// TIA Portal V20 export
// export: Created 2025-12-01T14:56:22.6342735Z, ExportSetting None, DisplayName Totally Integrated Automation Portal, DisplayVersion V20 Update 3, DisplayName TIA Portal Openness, DisplayVersion V20 Update 3, DisplayName TIA Portal Version Control Interface, DisplayVersion V20 Update 3, DisplayName STEP 7 Professional, DisplayVersion V20 Update 3, DisplayName STEP 7 Safety, DisplayVersion V20 Update 2, DisplayName WinCC Basic/Comfort/Advanced, DisplayVersion V20 Update 3, DisplayName WinCC Professional, DisplayVersion V20 Update 3, DisplayName WinCC Unified, DisplayVersion V20 Update 3
TYPE "EstadosMesa_Transporte_Paletizador_NDD"
   STRUCT
      Etapas_Reset : Bool;   // Etapa MESA en RESET
      Etapa_Vacia : Bool;   // Etapa MESA VACIA
      Etapa_Cargada : Bool;   // Etapa MESA CARGADA
      Etapas_Carga_E1 : Bool;   // Etapa CARGANDO MESA por E1
      Etapas_Descarga_S1 : Bool;   // Etapa DESCARGANDO MESA por S1
      Etapas_Carga_E2 : Bool;   // Etapa CARGANDO MESA por E2
      Etapas_Descarga_S2 : Bool;   // Etapa DESCARGANDO MESA por S2
      Etapas_Bloqueo : Bool;   // Etapa de BLOQUEO
      Descarga_Act : Bool;   // Memoria de DESCARGA ACTIVA
      Etapas_Carga_E0 : Bool;   // Etapa CARGANDO MESA por E0
      Etapas_Carga_E3 : Bool;   // Etapa CARGANDO MESA por E3
      Etapas_Descarga_S3 : Bool;   // Etapa DESCARGANDO MESA por S3
      Etapas_Carga_E4 : Bool;   // Etapa CARGANDO MESA por E4
      Etapas_Descarga_S4 : Bool;   // Etapa DESCARGANDO MESA por S4
      Etapas_Descarga_S0 : Bool;   // Etapa DESCARGANDO MESA por S0
      Manual : Bool;   // MESA EN MANUAL
      Err_Termico_E1_E3 : Bool;   // 01. TERMICO E1 E3
      Err_Termico_E2_E4 : Bool;   // 02. TERMICO E2 E4
      Err_Termico_Giro : Bool;   // 03. TERMICO GIRO
      Err_Mesa_Ocupada : Bool;   // 04. MESA OCUPADA
      Err_Perdida_PHs : Bool;   // 05. PERDIDA FOTOCELULA
      Err_TOut_Avance_E1_E3 : Bool;   // 06. TIMER TOUT Avance E1 E3
      Err_TOut_Retroceso_E1_E3 : Bool;   // 07. TIMER TOUT Retroceso E1 E3
      Err_TOut_Avance_E2_E4 : Bool;   // 08. TIMER TOUT Avance E2 E4
      Err_TOut_Retroceso_E2_E4 : Bool;   // 09. TIMER TOUT Retroceso E2 E4
      Err_TOut_Subir_TP_E1_E3 : Bool;   // 10. TIMER TOUT SUBIR TOPE E1 E3
      Err_TOut_Bajar_TP_E1_E3 : Bool;   // 11. TIMER TOUT BAJADA TOPE E1 E3
      Err_TOut_Subir_TP_E2_E4 : Bool;   // 12. TIMER TOUT SUBIDA TOPE E2 E4
      Err_TOut_Bajar_TP_E2_E4 : Bool;   // 13. TIMER TOUT BAJADA TOPE E2 E4
      Err_TOut_Bajada : Bool;   // 14. TIMER TOUT DE BAJADA DEL TRANSFER O MAQUETA
      Err_TOut_Subida : Bool;   // 15. TIMER TOUT DE SUBIDA DEL TRANSFER O MAQUETA
      Err_FTF_Sin_LibPHS_S1 : Bool;   // 16. FIN TRANSFER. SIN LIBERAR FOTOCELULA S1
      Err_FTF_Sin_LibPHS_S2 : Bool;   // 17. FIN TRANSFER. SIN LIBERAR FOTOCELULA S2
      Err_FTF_Sin_LibPHS_S3 : Bool;   // 18. FIN TRANSFER. SIN LIBERAR FOTOCELULA S3
      Err_FTF_Sin_LibPHS_S4 : Bool;   // 19. FIN TRANSFER. SIN LIBERAR FOTOCELULA S4
      Err_Salida_Lateral : Bool;   // 20. SALIDA LATERAL
      Err_Protusion : Bool;   // 21. PROTUSION
      Err_Interlock_Entrada : Bool;   // 22. INTERLOCK DE ENTRADA CON STV o VTD
      Err_Interlock_Salida : Bool;   // 23. INTERLOCK DE SALIDA CON STV o VTD
      Err_SegDescenso_EL : Bool;   // 24. DETECTOR DE DEGURIDAD EN DESCENSO DE LA MESA ELEVADORA
      Err_Tout_Giro : Bool;   // 25. TIMER TOUT DEL GIRO
      Err_Tout_Sacar : Bool;   // 26. TIMER TOUT DE SACRA LAS GARRAS
      Err_Tout_Recoger : Bool;   // 27. TIMER TOUT DE RECOGER LAS GARRAS
      Err_Tout_pos_0 : Bool;   // 28. TIMER TOUT DEL GIRO A 0º
      Err_Tout_pos_90 : Bool;   // 29. TIMER TOUT DEL GIRO A 90º
      Err_pHs_Galibo : Bool;   // 30. ERROR DE FOCELULAS DE GALIBO
      Err_DetectorTRANSFER : Bool;   // 31. ERROR DE DETECCION DEL TRANSFER ELECTRICO
      Err_Termico_elevacion : Bool;   // 32. ERROR TERMICO EN EL TRANSFER ELECTRICO
      Err_Nodo_SSCC : Bool;   // 33. ERROR PERDIDA NODO DEL SCANNER
      Err_SSCC_LectPorcentaje : Bool;   // 34. ERROR PORCENTAJE DE LECTURAS DE ESCANNER
      Err_SSCC_LectConsecutiva : Bool;   // 35. ERROR LECTURAS DE ESCANER CONSECUTICAS
      Err_MaquinaAsociada : Bool;   // 36. ERROR MAQUINA ASOCIADA A LA MESA
      Err_Extradimensiones : Bool;   // 37. ERROR PALETA FLEJADA
      Err_EnviadoPorJDT : Bool;   // 38. ERROR ENVIADO POR EL JDT
      Err_DatosPLC : Bool;   // 39. ERROR DE DATOS DEL PLC
      Error_Mx : Bool;   // Marca General Error
      En_Termico1 : Bool;   // Entrada de TERMICO 1
      En_Termico2 : Bool;   // Entrada de TERMICO 2
      En_PHS_1 : Bool;   // Entrada de FOTOCELULA 1
      En_PHS_2 : Bool;   // Entrada de FOTOCELULA 2
      En_Transfer_UP : Bool;   // Entrada TRANSFER/MAQUETA/MESA ELEVADORA ARRIBA
      En_Transfer_DOWN : Bool;   // Entrada TRANSFER/MAQUETA/MESA ELEVADORA ABAJO
      En_Tope1_UP : Bool;   // Entrada TOPE 1 ARRIBA
      En_Tope1_DOWN : Bool;   // Entrada TOPE 1 ABAJO
      En_Tope2_UP : Bool;   // Entrada TOPE 2 ARRIBA
      En_Tope2_DOWN : Bool;   // Entrada TOPE 2 ABAJO
      En_PHS_3 : Bool;   // Entrada de FOTOCELULA 3
      En_PHS_4 : Bool;   // Entrada de FOTOCELULA 4
      En_PHS_5 : Bool;   // Entrada de FOTOCELULA 5
      En_Giro_270 : Bool;   // …
      En_pHs_Prot1 : Bool;   // Entrada PROTUSION 1
      En_Detector_carretilla : Bool;   // Entrada detector de carretilla
      En_Giro_0 : Bool;   // Entrada Giro pos 0
      En_Giro_90 : Bool;   // Entrada Giro pos 90
      En_Giro_180 : Bool;   // Entrada Giro pos 180
      En_pHs_Prot2 : Bool;   // Entrada PROTUSION 2
      En_pHs_Prot3 : Bool;   // Entrada PROTUSION 3
      En_pHs_Prot4 : Bool;   // Entrada PROTUSION 4
      En_Empuj_Extendido : Bool;   // Entrada Empujador extendido (cilindro)
      En_Empuj_Recogido : Bool;   // Entrada Empujador recogido (cilindro)
      Sa_Rod_Avance : Bool;   // Salida AVANCE Rodillos
      Sa_Rod_Retroc : Bool;   // Salida RETROCEDE Rodillos
      Sa_Cad_Avance : Bool;   // Salida AVANCE Cadenas
      Sa_Cad_Retroc : Bool;   // Salida RETROCEDE Cadenas
      Sa_Trans_Sub : Bool;   // Salida SUBIR Transfer/Maqueta/mesa elevadora
      Sa_Trans_Baj : Bool;   // Salida BAJAR Transfer/Maqueta/mesa elevadora
      Sa_Tope1_Sub : Bool;   // Salida SUBIR Tope1
      Sa_Tope1_Baj : Bool;   // Salida BAJAR Tope1
      Sa_Tope2_Sub : Bool;   // Salida SUBIR Tope2
      Sa_Tope2_Baj : Bool;   // Salida BAJAR Tope2
      Sa_Giro_0 : Bool;   // Salida Girar a 0 grados
      Sa_Giro_90 : Bool;   // Salida Girar a 90 grados
      Sa_Giro_180 : Bool;   // Salida Girar a 180 grados
      Sa_Extender_Empujador : Bool;   // Salida extender_empujador (cilindro)
      Sa_Recoger_Empujador : Bool;   // Salida recoger empujador (cilindro)
      Sa_Giro_270 : Bool;   // ...
      Byte12_bit0 : Bool;   // ...
      Byte12_bit1 : Bool;   // ...
      Fin_VI : Bool;   // Fin de Vehiculo
      Paro_Blando : Bool;   // Mesa en paro blando
      Byte12_bit4 : Bool;   // ...
      Byte12_bit5 : Bool;   // ...
      Byte12_bit6 : Bool;   // ...
      Byte12_bit7 : Bool;   // ...
      Bumper_Mesa_Elevadora : Bool;   // ...
      Phs_Seguridad_1 : Bool;   // ...
      Phs_Seguridad_2 : Bool;   // ...
      Byte13_bit3 : Bool;   // ...
      Byte13_bit4 : Bool;   // ...
      Byte13_bit5 : Bool;   // ...
      Byte13_bit6 : Bool;   // …
      Byte13_bit7 : Bool;   // …
      Byte14_bit0 : Bool;   // …
      Byte14_bit1 : Bool;   // …
      Byte14_bit2 : Bool;   // ...
      Byte14_bit3 : Bool;   // ...
      Byte14_bit4 : Bool;   // ...
      Byte14_bit5 : Bool;   // ...
      Byte14_bit6 : Bool;   // ...
      Byte14_bit7 : Bool;   // ...
      pHs_CorteVelocidad : Bool;   // ...
      pHs_Seguridad : Bool;   // ...
      Byte15_bit2 : Bool;   // ...
      Byte15_bit3 : Bool;   // ...
      Byte15_bit4 : Bool;   // ...
      Byte15_bit5 : Bool;   // ...
      Byte15_bit6 : Bool;   // ...
      Byte15_bit7 : Bool;   // ...
   END_STRUCT;
END_TYPE
